// TIA Portal V19 export
TYPE "ValveSts"
// stored: Access Published
   STRUCT
      AlarmPresence : Bool;   // Status: Alarm rest / Cumulative alarm presence
      RestPermit : Bool;   // Status: Rest is permitted / Rest permitted
      RestInProgress : Bool;   // Status: Rest is in progress / Rest command in progress
      IsAtRest : Bool;   // Status: Valve is at rest / Valve is at Rest
      WorkPermit : Bool;   // Status: Work is permitted / Work permitted
      WorkInProgress : Bool;   // Status: Work is in progress / Work command in progress
      IsAtWork : Bool;   // Status: Valve is at work / Valve is at Work
      StandStill : Bool;   // Status: Is Standstill / Valve is standstill
   END_STRUCT;
END_TYPE
